// TIA Portal V18 export
// export: Created 2025-12-01T17:51:10.7823967Z, ExportSetting None, DisplayName Totally Integrated Automation Portal, DisplayVersion V18 Update 5, DisplayName TIA Portal Openness, DisplayVersion V18 Update 5, DisplayName TIA Portal Teamcenter Gateway, DisplayVersion V18, DisplayName TIA Portal Version Control Interface, DisplayVersion V18, DisplayName STEP 7 Professional, DisplayVersion V18 Update 5, DisplayName STEP 7 Safety, DisplayVersion V18, DisplayName WinCC Professional, DisplayVersion V18 Update 5
DATA_BLOCK "Axis_FB_DB"   // DB2200
// stored: AutoNumber false, InstanceOfName Axis_FB, InstanceOfType FB
"Axis_FB"
   // VAR RETAIN
   //    IAI_Axis { S7_SetPoint := 'True'} : Array[1..3] of "IAI_BASE_FB";
   // END_VAR
BEGIN
   // IAI_Axis[1] : Z轴
   // IAI_Axis[2] : X轴
   // IAI_Axis[3] : Y轴
   // IAI_Axis[1].Par.PosCode : Z轴
   // IAI_Axis[2].Par.PosCode : X轴
   // IAI_Axis[3].Par.PosCode : Y轴
END_DATA_BLOCK
